Staubli VAL3: jCadClean.pgx

program jCadClean()
  local num l_ni
begin
  //  nTotalPoints=size(jCad)
  //  if nTotalPoints<=1
  //    //          //no point
  //    //          io:socket="(RBINIT)"
  //  else
  //    //delete points
  //    for l_ni=nTotalPoints to 2 step -1
  //      $ddel(jCad,nTotalPoints-1)
  //      nTotalPoints=nTotalPoints-1
  //      nScrPts=nTotalPoints
  //      call hmi_refreshmain()
  //    endFor
  //    wait(nTotalPoints==1)
  //    //          io:socket="(RBINIT)"
  //  endIf
end
